(* IEC 61131-3 sources: LASAL/Class/Invert, 1 file *)

(* ---- Invert.st ---- *)
(*!
<Class
	Name               = "Invert"
	Revision           = "0.0"
	RealtimeTask       = "false"
	CyclicTask         = "false"
	BackgroundTask     = "false"
	Sigmatek           = "false"
	OSInterface        = "false"
	HighPriority       = "false"
	Automatic          = "false"
	UpdateMode         = "Prescan"
	SharedCommandTable = "true"
	Objectsize         = "(284,120)">
	<Channels>
		<Server Name="fIn" Visualized="false" Initialize="false" WriteProtected="false" Retentive="false"/>
		<Server Name="Sign" Visualized="false" Initialize="false" WriteProtected="false" Retentive="File"/>
		<Client Name="fOut" Required="true" Internal="false"/>
	</Channels>
</Class>
*)
Invert : CLASS
  //Servers:
	fIn 	: SvrChCmd_DINT;
	Sign 	: SvrCh_DINT;
  //Clients:
	fOut 	: CltCh_DINT;
  //Variables:
  //Functions:

	FUNCTION VIRTUAL GLOBAL fIn::Write
		VAR_INPUT
			input (EAX) 	: DINT;
		END_VAR
		VAR_OUTPUT
			result (EAX) 	: DINT;
		END_VAR;
  //Tables:
	FUNCTION @STD
		VAR_OUTPUT
			ret_code	: CONFSTATES;
		END_VAR;
	FUNCTION GLOBAL TAB @CT_;
END_CLASS;

FUNCTION VIRTUAL GLOBAL Invert::fIn::Write
	VAR_INPUT
		input (EAX) 	: DINT;
	END_VAR
	VAR_OUTPUT
		result (EAX) 	: DINT;
	END_VAR

	fIn := input;
  fOut:=fIn*sign;
  fOut.Write(input:=fOut);
	result := fIn;

END_FUNCTION
